{attribute 'reflection'} 
FUNCTION_BLOCK FB_Heater IMPLEMENTS I_SysModules
VAR
	lrCurrentTemp : LREAL := 72.0;
	sStatus		  : STRING := 'Heating...';
	
	{attribute 'instance-path'} 
    {attribute 'noinit'} 
    sPath : STRING; 
END_VAR

METHOD accept
VAR_INPUT
	iVisitor : I_Visitor;
END_VAR
iVisitor.visitHeater(THIS^);
END_METHOD

PROPERTY pPath : STRING
GET
pPath := THIS^.sPath;
END_GET
END_PROPERTY

PROPERTY pStatus : STRING
GET
pStatus := THIS^.sStatus;
END_GET
END_PROPERTY

PROPERTY pTemp : LREAL
GET
pTemp := THIS^.lrCurrentTemp;
END_GET
END_PROPERTY

END_FUNCTION_BLOCK

(* stored: Version 1.1.0.1, ProductVersion 3.1.4024.12
   POU FB_Heater: Id {1f9185b3-e3ce-4e45-a157-5f473ef16cdb}, SpecialFunc None
   Method accept: Id {219d35d4-b079-4f05-9455-c0331a726c1f}
   Property pPath: Id {c56d2ee8-fc14-4b91-b359-971aabafdd9d}
   Get Get: Id {83602bde-edda-4d14-a40e-0792d3b73791}
   Property pStatus: Id {dc6254ab-ed74-4917-a741-e37379d1bf61}
   Get Get: Id {9d847b6c-a219-476a-8d6e-049d01b68814}
   Property pTemp: Id {b9c50f6e-9cc5-4b5b-b278-c291c84a7d2b}
   Get Get: Id {1d9ebdfa-04e5-4b57-9efe-a4de3f893017} *)
